TYPE ADSCommunicationInterface :
STRUCT
	LocalAMSNetId	:	STRING;
	DeviceIpAddress	:	STRING;
	RuntimeStatus	:	STRING;
	HeartbeatPLC	:	BOOL;
	HeartbeatHMI	:	BOOL;
END_STRUCT
END_TYPE

(* stored: Version 1.1.0.1
   DUT ADSCommunicationInterface: Id {5538274f-e4c9-442d-b829-0b51909b43a9} *)
